(* CODESYS project Software_CLP.project

Project tree, tasks and I/O mapping:
  Device : CODESYS Control Win V3, 3S - Smart Software Solutions GmbH, order no. 305021, version 3.5.11.30
    application Application
      libraries: Standard, * (System)
      task MainTask (cyclic, interval t#20ms, priority 1) calls PLC_PRG
      task VISU_TASK (cyclic, interval 100 ms, priority 31) calls VisuElems.Visu_Prg
      program PLC_PRG [LD]
      visualisation Visualization
      Symbols
  libraries: VisuSymbols, 3.5.10.0 (System)
  text list GlobalTextList
*)

// Device/Application/PLC_PRG
PROGRAM PLC_PRG
VAR
	I0: BYTE;
	Q0: BYTE;
	M0: BYTE;
	QB1: BOOL;
	IB0: BOOL;
END_VAR

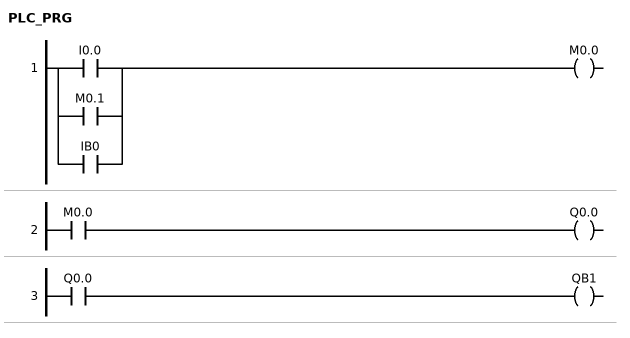
// NETWORK 1
M0.0 := I0.0 OR M0.1 OR IB0;

// NETWORK 2
Q0.0 := M0.0;

// NETWORK 3
QB1 := Q0.0;

END_PROGRAM

// Device/Application/Visualization
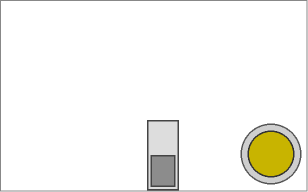
VISUALIZATION Visualization  // 308x192
    DipSwitch (128,120 70x70), variable: PLC_PRG.M0.1, behaviour: TOGGLE, style: Switch-DipSwitch-Gray
    Lamp1 (236,119 70x70), variable: PLC_PRG.Q0.0, style: Lamp-Lamp1-Yellow
END_VISUALIZATION
